FUNCTION_BLOCK I_GBSD (* Ground-based Speed and Distance GBSD *)
  (* Standard: ISO 11783-7; Classification: PGN 65097; Function: Ground-based Speed and Distance GBSD; Description: Copyright (c) 2024 HR Agrartechnik GmbH This program and the accompanying materials are made available under the terms of the Eclipse Public License 2.0 which is available at https://www.eclipse.org/legal/epl-2.0/ SPDX-License-Identifier: EPL-2.0 Message normally sent by the Tractor ECU on the implement bus on construction and agricultural implements providing to connected systems the current measured ground speed (also includes a free-running distance counter and an indication of the direction of travel). Accuracies of both wheel-based and ground-based sources can be speed-dependent and degrade at low speeds. Wheel-based information might not be updated at the 100 ms rate at low speeds. https://docs.ms-muc-docs.de/projects/isobus-other-docs/de/latest/PGN/PGN_65097.html *)
  (* Version 1.0, 2024-07-09, Franz Höpfinger, HR Agrartechnik GmbH *)
  PACKAGE isobus::tecu;
  IMPORT eclipse4diac::core::TypeHash;
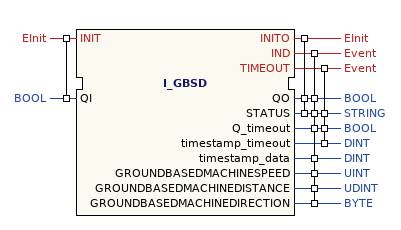
  EVENT_INPUT
    INIT : EInit WITH QI; (* Service Initialization *)
  END_EVENT
  EVENT_OUTPUT
    INITO : EInit WITH QO, STATUS; (* Initialization Confirm *)
    IND WITH QO, timestamp_data, GROUNDBASEDMACHINESPEED, GROUNDBASEDMACHINEDISTANCE, GROUNDBASEDMACHINEDIRECTION, STATUS, Q_timeout; (* Indication from Resource *)
    TIMEOUT WITH timestamp_timeout, STATUS, Q_timeout;
  END_EVENT
  VAR_INPUT
    QI : BOOL; (* Event Input Qualifier *)
  END_VAR
  VAR_OUTPUT
    QO : BOOL; (* Event Output Qualifier *)
    STATUS : STRING;
    Q_timeout : BOOL;
    timestamp_timeout : DINT;
    timestamp_data : DINT;
    GROUNDBASEDMACHINESPEED : UINT := UINT#16#FFFF; (* Ground-based machine speed (see Attributes for Details) *) {SET_ATTRIBUTE(SPN, 1859)} {SET_ATTRIBUTE(SP_Name, 'Ground-based machine speed')} {SET_ATTRIBUTE(SP_Position_In_PG, '1-2')} {SET_ATTRIBUTE(SP_Length, 16)} (* 16 bits *) {SET_ATTRIBUTE(Scaling, '0.001 m/s per bit')} {SET_ATTRIBUTE(Offset, )} {SET_ATTRIBUTE(Link, 'https://docs.ms-muc-docs.de/projects/isobus-other-docs/de/latest/PGN/PGN_65097.html#spn-1859-ground-based-machine-speed')}
    GROUNDBASEDMACHINEDISTANCE : UDINT := UDINT#16#FFFFFFFF; (* Ground-based machine distance (see Attributes for Details) *) {SET_ATTRIBUTE(SPN, 1860)} {SET_ATTRIBUTE(SP_Name, 'Ground-based machine distance')} {SET_ATTRIBUTE(SP_Position_In_PG, '3-6')} {SET_ATTRIBUTE(SP_Length, 32)} (* 32 bits *) {SET_ATTRIBUTE(Scaling, '0.001 m/bit')} {SET_ATTRIBUTE(Offset, )} {SET_ATTRIBUTE(Link, 'https://docs.ms-muc-docs.de/projects/isobus-other-docs/de/latest/PGN/PGN_65097.html#spn-1860-ground-based-machine-distance')}
    GROUNDBASEDMACHINEDIRECTION : BYTE := BYTE#16#FF; (* Ground-based machine direction (see Attributes for Details) *) {SET_ATTRIBUTE(SPN, 1861)} {SET_ATTRIBUTE(SP_Name, 'Ground-based machine direction')} {SET_ATTRIBUTE(SP_Position_In_PG, '8.1')} {SET_ATTRIBUTE(SP_Length, 2)} (* 2 bits *) {SET_ATTRIBUTE(Scaling, '4 states/2 bit')} {SET_ATTRIBUTE(Offset, )} {SET_ATTRIBUTE(Link, 'https://docs.ms-muc-docs.de/projects/isobus-other-docs/de/latest/PGN/PGN_65097.html#spn-1861-ground-based-machine-direction')}
  END_VAR
END_FUNCTION_BLOCK
